// TIA Portal V17 export
// export: Created 2024-01-13T10:45:56.6812483Z, ExportSetting WithDefaults, DisplayName Totally Integrated Automation Portal, DisplayVersion V17, DisplayName TIA Portal Openness, DisplayVersion V17, DisplayName TIA Portal Version Control Interface, DisplayVersion V17, DisplayName STEP 7 Professional, DisplayVersion V17, DisplayName STEP 7 Safety, DisplayVersion V17, DisplayName WinCC Advanced, DisplayVersion V17
FUNCTION_BLOCK "2.9 Crane ID Monitor"   // FB19, LAD
{ S7_Optimized_Access := 'TRUE' }
VERSION : 0.1
// stored: AutoNumber false, IsIECCheckEnabled false, IsRetainMemResEnabled false, MemoryReserve 100, SetENOAutomatically false, UDAEnableTagReadback false
   VAR
      "Crane ID Check Fault" { S7_SetPoint := 'True'} : "FB2502:Conditional Check";
   END_VAR
   VAR_TEMP   // added for the SCL form of the ladder/FBD networks
      _w1 : Bool;
      _s5time1 : S5Time;
   END_VAR
BEGIN

REGION Network 1: Crane ID Number Check Fault
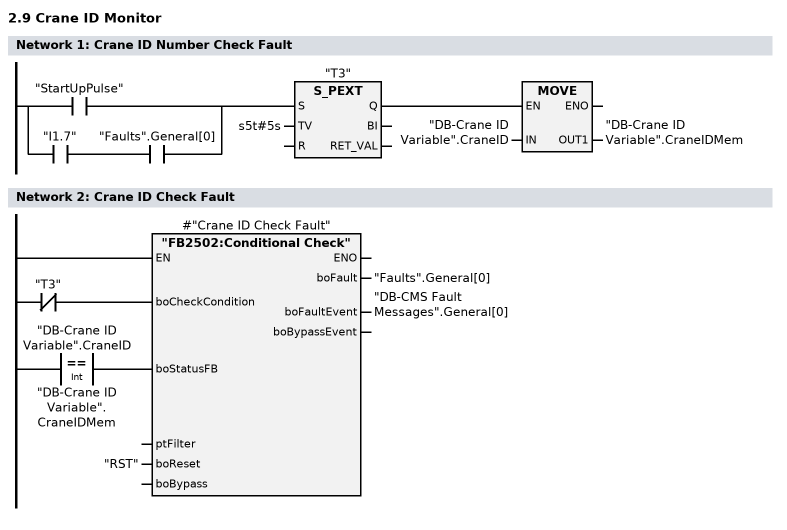
   RUNG wire#powerrail
      Contact( "StartUpPulse" )
      wire#w1
      S_PEXT(T_NO := "T3", TV := s5t#5s, R :=, BI =>, RET_VAL =>)
      Move(in := "DB-Crane ID Variable".CraneID, out1 => "DB-Crane ID Variable".CraneIDMem)
   END_RUNG
   RUNG wire#powerrail
      Contact( "I1.7" )
      Contact( "Faults".General[0] )
   END_RUNG wire#w1
   // the same network as SCL:
   #_s5time1 := S_PEXT(T_NO := "T3",
                       S := "StartUpPulse" OR ("I1.7" AND "Faults".General[0]),
                       TV := s5t#5s,
                       Q => #_w1);
   IF #_w1 THEN "DB-Crane ID Variable".CraneIDMem := "DB-Crane ID Variable".CraneID; END_IF;
END_REGION

REGION Network 2: Crane ID Check Fault
   RUNG wire#powerrail
      #"Crane ID Check Fault"(boCheckCondition := wire#w1, boStatusFB := wire#w2, ptFilter :=, boReset := "RST", boBypass :=, boFault => "Faults".General[0], boFaultEvent => "DB-CMS Fault Messages".General[0], boBypassEvent =>)
   END_RUNG
   RUNG wire#powerrail
      I_Contact( "T3" )
   END_RUNG wire#w1
   RUNG wire#powerrail
      { S7_Templates := "SrcType := Int" } EQ_Contact(in1 := "DB-Crane ID Variable".CraneID, in2 := "DB-Crane ID Variable".CraneIDMem)
   END_RUNG wire#w2
   // the same network as SCL:
   #"Crane ID Check Fault"(boCheckCondition := NOT "T3",   // "FB2502:Conditional Check"
                           boStatusFB := "DB-Crane ID Variable".CraneID = "DB-Crane ID Variable".CraneIDMem,
                           boReset := "RST",
                           boFault => "Faults".General[0],
                           boFaultEvent => "DB-CMS Fault Messages".General[0]);
END_REGION
END_FUNCTION_BLOCK
